SYSTEM test
  (* Version 1.0, 2023-10-23, franz *)
  APPLICATION App_functions
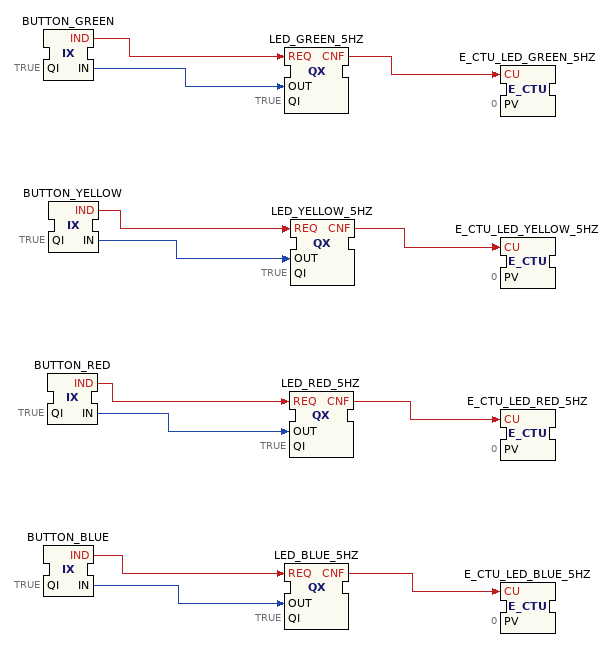
    FBS
      BUTTON_RED : IX(QI := TRUE);
      BUTTON_YELLOW : IX(QI := TRUE);
      BUTTON_BLUE : IX(QI := TRUE);
      LED_YELLOW_5HZ : QX(QI := TRUE);
      LED_BLUE_5HZ : QX(QI := TRUE);
      LED_RED_5HZ : QX(QI := TRUE);
      BUTTON_GREEN : IX(QI := TRUE);
      LED_GREEN_5HZ : QX(QI := TRUE);
      E_CTU_LED_GREEN_5HZ : E_CTU(PV := 0);
      E_CTU_LED_YELLOW_5HZ : E_CTU(PV := 0);
      E_CTU_LED_RED_5HZ : E_CTU(PV := 0);
      E_CTU_LED_BLUE_5HZ : E_CTU(PV := 0);
    END_FBS
    EVENT_CONNECTIONS
      BUTTON_RED.IND TO LED_RED_5HZ.REQ;
      BUTTON_YELLOW.IND TO LED_YELLOW_5HZ.REQ;
      BUTTON_BLUE.IND TO LED_BLUE_5HZ.REQ;
      BUTTON_GREEN.IND TO LED_GREEN_5HZ.REQ;
      LED_GREEN_5HZ.CNF TO E_CTU_LED_GREEN_5HZ.CU;
      LED_YELLOW_5HZ.CNF TO E_CTU_LED_YELLOW_5HZ.CU;
      LED_RED_5HZ.CNF TO E_CTU_LED_RED_5HZ.CU;
      LED_BLUE_5HZ.CNF TO E_CTU_LED_BLUE_5HZ.CU;
    END_CONNECTIONS
    DATA_CONNECTIONS
      BUTTON_RED.IN TO LED_RED_5HZ.OUT;
      BUTTON_YELLOW.IN TO LED_YELLOW_5HZ.OUT;
      BUTTON_BLUE.IN TO LED_BLUE_5HZ.OUT;
      BUTTON_GREEN.IN TO LED_GREEN_5HZ.OUT;
    END_CONNECTIONS
  END_APPLICATION
  APPLICATION App_mapping
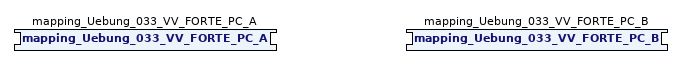
    SUBAPPS
      mapping_Uebung_033_VV_FORTE_PC_A : mapping_Uebung_033_VV_FORTE_PC_A;
      mapping_Uebung_033_VV_FORTE_PC_B : mapping_Uebung_033_VV_FORTE_PC_B;
    END_SUBAPPS
  END_APPLICATION
  DEVICE FORTE_PC_A : FORTE_PC(MGR_ID := C_PC_A (* Device manager socket ID *))
    {SET_ATTRIBUTE(Profile, HOLOBLOC)}
    {SET_ATTRIBUTE(FBType, GEN_E_MUX, F_LT, F_INT_AS_WSTRING, UT_ButtonMapping_UP, F_LWORD_TO_WORD, F_TIME_IN_S_TO_UDINT, F_TAN, F_DINT_TO_UINT, F_BYTE_AS_STRING, F_ADD_DT_TIME, F_TIME_IN_US_TO_LREAL, F_INT_TO_UDINT, F_ADD_TOD_TIME, F_SUB_DT_DT, F_DT_TO_TOD, F_UINT_TO_BCD_WORD, F_UDINT_TO_REAL, UT_AuxiliaryInputMapping_Type_10_CombinedAnalog_LatchBool, F_REAL_TO_UDINT, F_WSTRING_AS_TIME, F_DWORD_TO_WORD, F_MUL, TEST_CONDITION, F_LE, GEN_SUBSCRIBE, F_LN, F_WSTRING_AS_BOOL, F_STRING_AS_UDINT, F_DWORD_AS_WSTRING, GEN_OR, E_CYCLE, F_STRING_AS_BYTE, UT_ButtonMapping, F_LREAL_TO_SINT, F_STRING_AS_DINT, E_F_TRIG, F_LWORD_TO_UINT, F_INT_AS_STRING, E_RS, F_UINT_TO_WORD, F_WORD_TO_DINT, F_USINT_AS_WSTRING, UT_AuxiliaryInputMapping_Type_13_QuadratAnalog_Ret50perc, F_OR, F_STRING_AS_INT, F_WORD_TO_BYTE, F_LREAL_AS_WSTRING, F_TIME_IN_NS_TO_ULINT, F_WSTRING_AS_WORD, STEST_END, F_NE, F_LWORD_TO_ULINT, F_INT_TO_BYTE, F_INT_TO_DINT, F_ULINT_TO_LINT, F_DWORD_TO_UINT, DWORD2DWORD, UT_AuxiliaryInputMapping_Type_12_QuadratAnalog, F_TIME_IN_NS_TO_LINT, UT_NumericValueInputMapping, E_SELECT, F_MULTIME, F_USINT_TO_INT, F_DWORD_TO_UDINT, F_BYTE_TO_DI, F_UINT_TO_LWORD, Q_CtrlAudioSignal, F_SINT_TO_LWORD, GEN_F_MUX, USINT2USINT, Q_ChangeObjectLabel, F_LINT_TO_SINT, UT_AuxiliaryInputMapping_Type_01_Analog_0_100perc, F_WORD_TO_USINT, F_DWORD_TO_INT, F_LREAL_TO_REAL, Q_LockUnlockMask, F_LEFT, F_SINT_AS_WSTRING, F_BYTE_AS_WSTRING, F_TIME_IN_MS_TO_DINT, E_SR, F_UDINT_TO_BCD_DWORD, F_LWORD_AS_STRING, PUBLISH_1, GEN_XOR, F_DINT_TO_WORD, F_SUB_TOD_TIME, E_RESTART, E_PERMIT, TIME2TIME, F_UINT_TO_SINT, F_XOR, Q_ESC, F_SEL, F_ULINT_TO_LREAL, Q_ChangePolygonPoint, F_SINT_TO_LREAL, F_DINT_TO_SINT, E_TimeOut, Hutschienenmoped_XL_8_DI_LONG_PRESS_HOLD, F_BYTE_TO_UDINT, UT_AuxiliaryInputMapping_Type_04_Analog_Ret0perc, Q_Size, F_REPLACE, F_LINT_TO_USINT, SUBSCRIBE_1, signalprocessing__DualHysteresis, F_ABS, F_WORD_TO_LWORD, E_DELAY, GEN_ADD, Q_GraphicsContext, F_DINT_TO_USINT, F_REAL_AS_WSTRING, F_INT_TO_REAL, E_CTU, F_WSTRING_AS_SINT, Q_NumericValue, Q_ExecuteMacro, F_MOVE, F_WSTRING_TO_STRING, F_USINT_TO_LINT, F_DIV, E_CTD, F_UINT_TO_DWORD, F_LWORD_TO_LINT, F_ADD, F_BYTE_TO_LINT, F_TIME_IN_MS_TO_LREAL, F_LREAL_TO_UINT, F_ACOS, F_WSTRING_AS_LREAL, F_DWORD_TO_LINT, F_SHL, F_REAL_TO_ULINT, F_ULINT_TO_UINT, F_UDINT_TO_SINT, NVS_UDINT, F_SHR, UINT2UINT, F_WORD_TO_DWORD, F_INT_TO_LWORD, F_USINT_TO_UINT, Q_FontAttributes, F_INT_TO_ULINT, F_USINT_AS_STRING, GEN_CSV_WRITER, F_LINT_TO_WORD, F_UINT_TO_LREAL, F_SINT_TO_WORD, Q_ChangePolygonScale, Q_ExecuteExtendedMacro, F_STRING_TO_WSTRING, STRING2STRING, UT_AuxiliaryInputMapping_Type_00_Bool_Latched, F_LREAL_TO_DINT, F_SIN, F_UINT_TO_USINT, GetInstancePath, F_LREAL_AS_STRING, UT_AuxiliaryInputMapping_Type_08_DualBool_LatchedDown, F_DINT_TO_ULINT, F_REAL_TO_UINT, F_ULINT_TO_WORD, F_INT_TO_LINT, UT_ButtonMapping_HOLD, E_D_FF, F_STRING_AS_ULINT, F_ULINT_AS_STRING, F_INT_TO_DWORD, F_WORD_TO_LINT, F_UDINT_TO_INT, REAL2REAL, F_LREAL_TO_USINT, F_DINT_TO_LWORD, DEV_MGR, F_SINT_TO_UINT, E_CTUD, SET_STRUCT_VALUE, UT_SoftkeyMapping_UP, F_ULINT_AS_WSTRING, E_RDELAY, F_SINT_TO_ULINT, F_WSTRING_AS_LINT, Q_FillAttributes, UT_ButtonMapping_DOWN, Hutschienenmoped_XL_8_DI_DOWN, F_STRING_AS_LINT, F_LINT_TO_ULINT, UT_AuxiliaryInputMapping_Type_14_BidirectionalCounter, F_RIGHT, F_SINT_TO_INT, NVS_UINT, SINT2SINT, Q_ObjEnableDisable, F_UDINT_AS_STRING, F_TIME_IN_NS_TO_UDINT, F_LINT_TO_LWORD, F_LWORD_TO_UDINT, F_TRUNC, F_ULINT_TO_DWORD, F_STRING_AS_UINT, F_TIME_IN_MS_TO_UDINT, F_WSTRING_AS_UDINT, F_TIME_IN_S_TO_LREAL, F_DINT_AS_STRING, F_TIME_IN_NS_TO_DINT, E_TRAIN, OUT_ANY_CONSOLE, F_ULINT_TO_SINT, F_DINT_TO_LINT, F_UDINT_TO_DWORD, GEN_E_DEMUX, F_SQRT, F_UDINT_AS_WSTRING, F_LINT_AS_STRING, E_SR_RETRIG, Q_ListItem, F_WSTRING_AS_UINT, Q_ChildLocation, F_UINT_TO_INT, F_TIME_IN_S_TO_LINT, F_ULINT_TO_USINT, F_UINT_TO_REAL, F_LREAL_TO_LWORD, F_LINT_AS_WSTRING, UT_SoftkeyMapping, F_SINT_TO_LINT, Hutschienenmoped_XL_2_SERVO, F_MAX, F_LREAL_TO_INT, F_SINT_AS_STRING, F_UDINT_TO_LWORD, F_TIME_AS_WSTRING, Q_SetAudioVolume, INT2INT, UT_AuxiliaryInputMapping_Type_03_Analog_Ret50perc, F_DWORD_AS_STRING, F_BYTE_TO_ULINT, F_UDINT_TO_WORD, F_LINT_TO_UINT, F_TIME_IN_US_TO_ULINT, F_TIME_AS_STRING, F_COS, F_TIME_IN_NS_TO_LREAL, Q_ObjHideShow, F_REAL_TO_LINT, Hutschienenmoped_XL_8_DI_REPEAT, Hutschienenmoped_XL_1_LED_DO, F_USINT_TO_WORD, E_REND, F_ASIN, F_REAL_TO_INT, F_WORD_BCD_TO_UINT, F_STRING_AS_TIME, F_BYTE_TO_INT, EMB_RES, F_BYTE_TO_WORD, F_USINT_TO_LWORD, F_DWORD_TO_DINT, signalprocessing__FIELDBUS_PERCENT_TO_WORD, F_ULINT_TO_LWORD, F_USINT_TO_ULINT, GEN_SUBL, F_DWORD_TO_BYTE, UT_AuxiliaryInputMapping_Type_06_DualBool_BothNonLatched, F_DIVTIME, F_ROL, F_LWORD_TO_DINT, F_LWORD_AS_WSTRING, F_WORD_TO_SINT, F_LWORD_TO_BYTE, F_SEL_E_4, GEN_AND, F_AND, F_ROR, GEN_CLIENT, F_SEL_E_2, F_SEL_E_3, F_LREAL_TO_LINT, E_IMPULSE, WSTRING2WSTRING, F_WORD_TO_INT, F_UINT_TO_BYTE, F_UDINT_TO_UINT, F_SINT_TO_UDINT, F_UINT_TO_DINT, F_UINT_TO_UDINT, F_STRING_AS_WORD, F_DINT_TO_UDINT, F_WSTRING_AS_BYTE, E_SPLIT, F_DWORD_TO_LWORD, F_USINT_TO_SINT, E_STOPWATCH_T, F_ULINT_TO_BCD_LWORD, F_BYTE_BCD_TO_USINT, F_DWORD_TO_ULINT, F_BYTE_TO_SINT, F_STRING_AS_BOOL, F_WSTRING_AS_DINT, GEN_ARRAY2ARRAY, F_DT_TO_DATE, GEN_STRUCT_DEMUX, F_LEN, GEN_STRUCT_MUX, F_INT_TO_WORD, FB_RANDOM, F_LINT_TO_UDINT, Q_NumericValueAux, Q_LineAttributes, Hutschienenmoped_XL_8_DI_DOUBLE_CLICK, F_EXP, F_USINT_TO_DWORD, F_TIME_IN_MS_TO_ULINT, F_REAL_TO_SINT, Hutschienenmoped_XL_1_LED_PWM, F_INT_TO_USINT, F_EXPT, F_SUB, F_WSTRING_AS_ULINT, F_ULINT_TO_REAL, F_REAL_TO_LREAL, F_MID, F_BYTE_TO_UINT, F_BYTE_TO_DWORD, F_INT_TO_UINT, Q_BackgroundColourAux, F_DWORD_TO_REAL, F_DINT_TO_BYTE, F_SUB_TOD_TOD, SET_AT_INDEX, F_MIN, F_STRING_AS_LREAL, F_TIME_IN_S_TO_DINT, F_LREAL_TO_ULINT, F_STRING_AS_SINT, UT_SoftkeyMapping_HOLD, F_BYTE_TO_LWORD, F_UINT_AS_STRING, BOOL2BOOL, F_LINT_TO_INT, UT_SoftkeyMapping_DOWN, F_INSERT, F_SUB_DT_TIME, F_FIND, F_UDINT_TO_ULINT, F_WORD_AS_WSTRING, F_WORD_TO_UDINT, UT_AuxiliaryInputMapping_Type_07_DualBool_LatchedUp, F_DINT_TO_DWORD, F_UINT_AS_WSTRING, GEN_VALUES2ARRAY, GEN_ARRAY2VALUES, F_DINT_AS_WSTRING, F_TIME_IN_US_TO_UDINT, F_WORD_TO_UINT, Q_Priority, Q_ChildPosition, F_TIME_IN_US_TO_LINT, UT_AuxiliaryInputMapping_Type_11_QuadratBool_NonLatched, F_LINT_TO_DWORD, Q_GetAttribute, F_CONCAT, F_UDINT_TO_LINT, F_SUB_DATE_DATE, F_LWORD_TO_LREAL, F_LWORD_TO_INT, WORD2WORD, E_STOPWATCH, F_LIMIT, F_TIME_IN_S_TO_ULINT, F_LWORD_TO_USINT, F_WSTRING_AS_USINT, F_REAL_TO_DINT, F_DWORD_TO_USINT, Q_SelectColourMap, F_STRING_AS_DWORD, UT_AuxiliaryInputMapping_Type_09_CombinedAnalog_Ret50perc, Q_SoftKeyMask, E_MERGE, UT_AuxiliaryInputMapping_Type_05_DualBool_BothLatched, F_SINT_TO_DWORD, E_DEMUX, BYTE2BYTE, F_USINT_TO_BCD_BYTE, F_SINT_TO_DINT, Hutschienenmoped_XL_8_DO, F_UINT_TO_LINT, F_SINT_TO_BYTE, F_ATAN, F_LINT_TO_BYTE, F_BYTE_TO_USINT, F_ULINT_TO_UDINT, F_NOT, F_DINT_TO_INT, F_LINT_TO_DINT, F_DELETE, Q_ObjSelectInput, F_WSTRING_AS_DWORD, GEN_SERVER, Q_EndPoint, GEN_PUBL, Q_SelectActiveWorkingSet, F_UDINT_TO_LREAL, Hutschienenmoped_XL_8_DI, E_R_TRIG, F_REAL_AS_STRING, Q_ActiveMask, F_GE, F_LWORD_BCD_TO_ULINT, signalprocessing__FIELDBUS_WORD_TO_PERCENT, F_WSTRING_AS_INT, F_MUX_2, F_USINT_TO_UDINT, F_UINT_TO_ULINT, F_EQ, E_T_FF, F_USINT_TO_REAL, LREAL2LREAL, Hutschienenmoped_XL_8_DI_LONG_PRESS_START, F_MOD, E_RTimeOut, F_ULINT_TO_DINT, F_ULINT_TO_BYTE, GET_STRUCT_VALUE, GEN_PUBLISH, F_REAL_TO_DWORD, F_DWORD_BCD_TO_UDINT, F_INT_TO_LREAL, E_CTUD_UDINT, F_LWORD_TO_SINT, F_GT, F_LINT_TO_REAL, F_TIME_IN_MS_TO_LINT, F_STRING_AS_LWORD, F_SINT_TO_REAL, F_LOG, Hutschienenmoped_XL_8_AI, F_ULINT_TO_INT, F_DWORD_TO_SINT, F_REAL_TO_USINT, F_STRING_AS_REAL, E_SWITCH, F_LINT_TO_LREAL, UT_AuxiliaryInputMapping_Type_02_Bool_NonLatched, F_STRING_AS_USINT, F_SINT_TO_USINT, F_DINT_TO_REAL, DINT2DINT, Q_BackgroundColour, F_WSTRING_AS_LWORD, Q_Attribute, Hutschienenmoped_XL_8_DI_UP, F_WORD_TO_ULINT, F_WORD_AS_STRING, F_INT_TO_SINT, F_TIME_IN_US_TO_DINT, Hutschienenmoped_XL_8_DI_SINGLE_CLICK, F_CONCAT_DATE_TOD, GET_AT_INDEX, F_USINT_TO_LREAL, Q_StringValue, F_DINT_TO_LREAL, UDINT2UDINT, F_USINT_TO_BYTE, F_LWORD_TO_DWORD, F_LREAL_TO_UDINT, F_WSTRING_AS_REAL, F_UDINT_TO_DINT, F_UDINT_TO_BYTE, F_USINT_TO_DINT)} (* created during deployment *)
    RESOURCE EMB_RES : EMB_RES
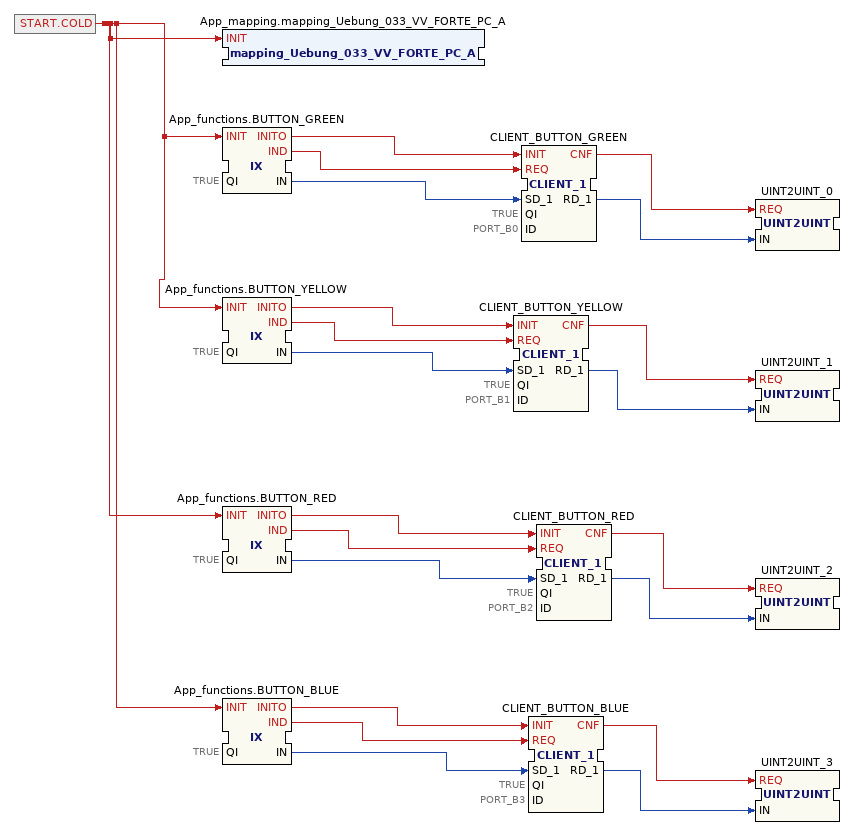
      FBS
        App_functions.BUTTON_BLUE : IX(QI := TRUE);
        App_functions.BUTTON_GREEN : IX(QI := TRUE);
        App_functions.BUTTON_RED : IX(QI := TRUE);
        App_functions.BUTTON_YELLOW : IX(QI := TRUE);
        CLIENT_BUTTON_GREEN : CLIENT_1(QI := TRUE, ID := PORT_B0);
        CLIENT_BUTTON_YELLOW : CLIENT_1(QI := TRUE, ID := PORT_B1);
        CLIENT_BUTTON_RED : CLIENT_1(QI := TRUE, ID := PORT_B2);
        CLIENT_BUTTON_BLUE : CLIENT_1(QI := TRUE, ID := PORT_B3);
        UINT2UINT_0 : UINT2UINT;
        UINT2UINT_1 : UINT2UINT;
        UINT2UINT_2 : UINT2UINT;
        UINT2UINT_3 : UINT2UINT;
      END_FBS
      SUBAPPS
        App_mapping.mapping_Uebung_033_VV_FORTE_PC_A : mapping_Uebung_033_VV_FORTE_PC_A;
      END_SUBAPPS
      EVENT_CONNECTIONS
        START.COLD TO App_mapping.mapping_Uebung_033_VV_FORTE_PC_A.INIT;
        App_functions.BUTTON_GREEN.INITO TO CLIENT_BUTTON_GREEN.INIT;
        App_functions.BUTTON_GREEN.IND TO CLIENT_BUTTON_GREEN.REQ;
        App_functions.BUTTON_YELLOW.INITO TO CLIENT_BUTTON_YELLOW.INIT;
        App_functions.BUTTON_YELLOW.IND TO CLIENT_BUTTON_YELLOW.REQ;
        App_functions.BUTTON_RED.INITO TO CLIENT_BUTTON_RED.INIT;
        App_functions.BUTTON_RED.IND TO CLIENT_BUTTON_RED.REQ;
        App_functions.BUTTON_BLUE.INITO TO CLIENT_BUTTON_BLUE.INIT;
        App_functions.BUTTON_BLUE.IND TO CLIENT_BUTTON_BLUE.REQ;
        CLIENT_BUTTON_GREEN.CNF TO UINT2UINT_0.REQ;
        CLIENT_BUTTON_YELLOW.CNF TO UINT2UINT_1.REQ;
        CLIENT_BUTTON_RED.CNF TO UINT2UINT_2.REQ;
        CLIENT_BUTTON_BLUE.CNF TO UINT2UINT_3.REQ;
        START.COLD TO App_functions.BUTTON_GREEN.INIT;
        START.COLD TO App_functions.BUTTON_YELLOW.INIT;
        START.COLD TO App_functions.BUTTON_RED.INIT;
        START.COLD TO App_functions.BUTTON_BLUE.INIT;
      END_CONNECTIONS
      DATA_CONNECTIONS
        App_functions.BUTTON_GREEN.IN TO CLIENT_BUTTON_GREEN.SD_1;
        App_functions.BUTTON_YELLOW.IN TO CLIENT_BUTTON_YELLOW.SD_1;
        App_functions.BUTTON_RED.IN TO CLIENT_BUTTON_RED.SD_1;
        App_functions.BUTTON_BLUE.IN TO CLIENT_BUTTON_BLUE.SD_1;
        CLIENT_BUTTON_RED.RD_1 TO UINT2UINT_2.IN;
        CLIENT_BUTTON_BLUE.RD_1 TO UINT2UINT_3.IN;
        CLIENT_BUTTON_YELLOW.RD_1 TO UINT2UINT_1.IN;
        CLIENT_BUTTON_GREEN.RD_1 TO UINT2UINT_0.IN;
      END_CONNECTIONS
    END_RESOURCE
  END_DEVICE
  DEVICE FORTE_PC_B : FORTE_PC(MGR_ID := C_PC_B (* Device manager socket ID *))
    {SET_ATTRIBUTE(Profile, HOLOBLOC)}
    RESOURCE EMB_RES : EMB_RES
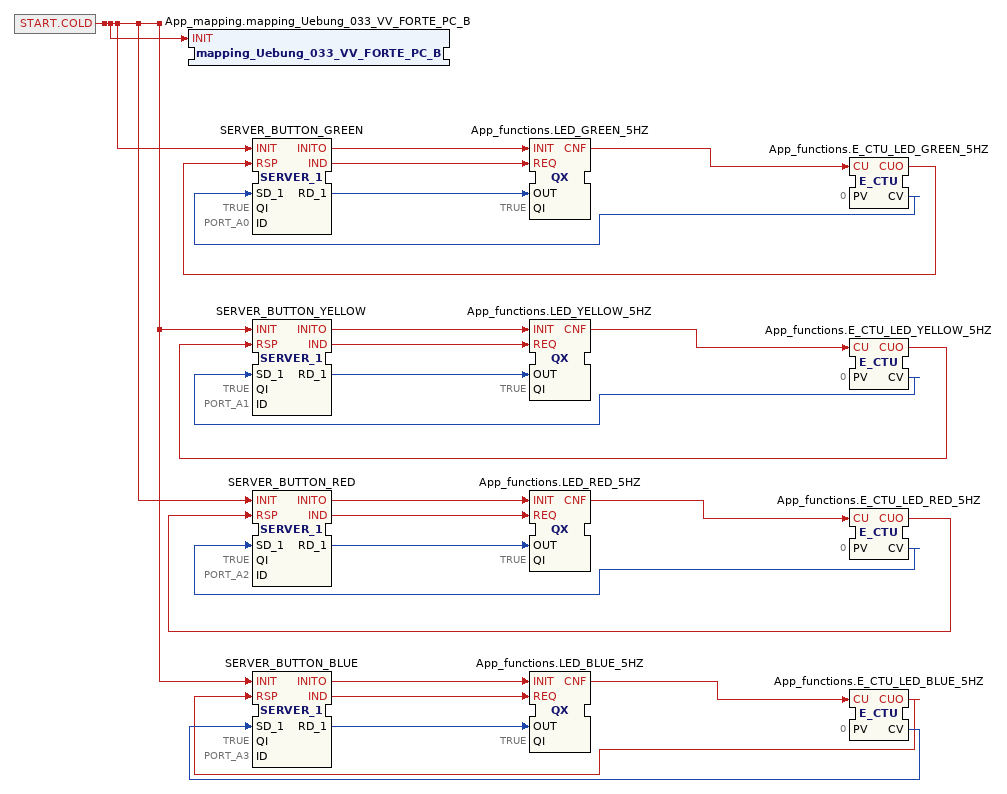
      FBS
        App_functions.LED_GREEN_5HZ : QX(QI := TRUE);
        App_functions.LED_RED_5HZ : QX(QI := TRUE);
        App_functions.LED_YELLOW_5HZ : QX(QI := TRUE);
        App_functions.LED_BLUE_5HZ : QX(QI := TRUE);
        SERVER_BUTTON_GREEN : SERVER_1(QI := TRUE, ID := PORT_A0);
        SERVER_BUTTON_RED : SERVER_1(QI := TRUE, ID := PORT_A2);
        SERVER_BUTTON_YELLOW : SERVER_1(QI := TRUE, ID := PORT_A1);
        SERVER_BUTTON_BLUE : SERVER_1(QI := TRUE, ID := PORT_A3);
        App_functions.E_CTU_LED_YELLOW_5HZ : E_CTU(PV := 0);
        App_functions.E_CTU_LED_RED_5HZ : E_CTU(PV := 0);
        App_functions.E_CTU_LED_GREEN_5HZ : E_CTU(PV := 0);
        App_functions.E_CTU_LED_BLUE_5HZ : E_CTU(PV := 0);
      END_FBS
      SUBAPPS
        App_mapping.mapping_Uebung_033_VV_FORTE_PC_B : mapping_Uebung_033_VV_FORTE_PC_B;
      END_SUBAPPS
      EVENT_CONNECTIONS
        START.COLD TO App_mapping.mapping_Uebung_033_VV_FORTE_PC_B.INIT;
        START.COLD TO SERVER_BUTTON_GREEN.INIT;
        SERVER_BUTTON_GREEN.INITO TO App_functions.LED_GREEN_5HZ.INIT;
        SERVER_BUTTON_GREEN.IND TO App_functions.LED_GREEN_5HZ.REQ;
        START.COLD TO SERVER_BUTTON_RED.INIT;
        SERVER_BUTTON_RED.INITO TO App_functions.LED_RED_5HZ.INIT;
        SERVER_BUTTON_RED.IND TO App_functions.LED_RED_5HZ.REQ;
        START.COLD TO SERVER_BUTTON_YELLOW.INIT;
        SERVER_BUTTON_YELLOW.INITO TO App_functions.LED_YELLOW_5HZ.INIT;
        SERVER_BUTTON_YELLOW.IND TO App_functions.LED_YELLOW_5HZ.REQ;
        START.COLD TO SERVER_BUTTON_BLUE.INIT;
        SERVER_BUTTON_BLUE.INITO TO App_functions.LED_BLUE_5HZ.INIT;
        SERVER_BUTTON_BLUE.IND TO App_functions.LED_BLUE_5HZ.REQ;
        App_functions.LED_YELLOW_5HZ.CNF TO App_functions.E_CTU_LED_YELLOW_5HZ.CU;
        App_functions.LED_RED_5HZ.CNF TO App_functions.E_CTU_LED_RED_5HZ.CU;
        App_functions.LED_GREEN_5HZ.CNF TO App_functions.E_CTU_LED_GREEN_5HZ.CU;
        App_functions.LED_BLUE_5HZ.CNF TO App_functions.E_CTU_LED_BLUE_5HZ.CU;
        App_functions.E_CTU_LED_BLUE_5HZ.CUO TO SERVER_BUTTON_BLUE.RSP;
        App_functions.E_CTU_LED_RED_5HZ.CUO TO SERVER_BUTTON_RED.RSP;
        App_functions.E_CTU_LED_YELLOW_5HZ.CUO TO SERVER_BUTTON_YELLOW.RSP;
        App_functions.E_CTU_LED_GREEN_5HZ.CUO TO SERVER_BUTTON_GREEN.RSP;
      END_CONNECTIONS
      DATA_CONNECTIONS
        SERVER_BUTTON_GREEN.RD_1 TO App_functions.LED_GREEN_5HZ.OUT;
        SERVER_BUTTON_RED.RD_1 TO App_functions.LED_RED_5HZ.OUT;
        SERVER_BUTTON_YELLOW.RD_1 TO App_functions.LED_YELLOW_5HZ.OUT;
        SERVER_BUTTON_BLUE.RD_1 TO App_functions.LED_BLUE_5HZ.OUT;
        App_functions.E_CTU_LED_GREEN_5HZ.CV TO SERVER_BUTTON_GREEN.SD_1;
        App_functions.E_CTU_LED_YELLOW_5HZ.CV TO SERVER_BUTTON_YELLOW.SD_1;
        App_functions.E_CTU_LED_RED_5HZ.CV TO SERVER_BUTTON_RED.SD_1;
        App_functions.E_CTU_LED_BLUE_5HZ.CV TO SERVER_BUTTON_BLUE.SD_1;
      END_CONNECTIONS
    END_RESOURCE
  END_DEVICE
  MAPPINGS
    App_mapping.mapping_Uebung_033_VV_FORTE_PC_A ON FORTE_PC_A.EMB_RES;
    App_functions.BUTTON_BLUE ON FORTE_PC_A.EMB_RES;
    App_functions.BUTTON_RED ON FORTE_PC_A.EMB_RES;
    App_functions.BUTTON_YELLOW ON FORTE_PC_A.EMB_RES;
    App_functions.LED_RED_5HZ ON FORTE_PC_B.EMB_RES;
    App_functions.LED_YELLOW_5HZ ON FORTE_PC_B.EMB_RES;
    App_functions.LED_BLUE_5HZ ON FORTE_PC_B.EMB_RES;
    App_mapping.mapping_Uebung_033_VV_FORTE_PC_B ON FORTE_PC_B.EMB_RES;
    App_functions.LED_GREEN_5HZ ON FORTE_PC_B.EMB_RES;
    App_functions.BUTTON_GREEN ON FORTE_PC_A.EMB_RES;
    App_functions.E_CTU_LED_YELLOW_5HZ ON FORTE_PC_B.EMB_RES;
    App_functions.E_CTU_LED_RED_5HZ ON FORTE_PC_B.EMB_RES;
    App_functions.E_CTU_LED_GREEN_5HZ ON FORTE_PC_B.EMB_RES;
    App_functions.E_CTU_LED_BLUE_5HZ ON FORTE_PC_B.EMB_RES;
  END_MAPPINGS
  SEGMENTS
    Ethernet : Ethernet;
  END_SEGMENTS
  LINKS
    FORTE_PC_A => Ethernet;
    FORTE_PC_B => Ethernet;
  END_LINKS
END_SYSTEM
